FUNCTION_BLOCK basicFalhaFeedback (* Basic Function Block Type *)
  (* Standard: 61499-2 *)
  (* Version 0.0, 14/01/2026, Schneider Electric, Template *)
  PACKAGE Hidryco.HidrycoLib;
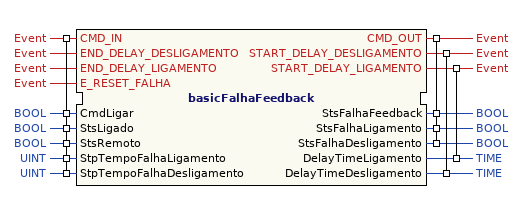
  EVENT_INPUT
    CMD_IN WITH StpTempoFalhaLigamento, StpTempoFalhaDesligamento, StsRemoto, CmdLigar, StsLigado;
    END_DELAY_DESLIGAMENTO; (* Normal Execution Request *)
    END_DELAY_LIGAMENTO;
    E_RESET_FALHA;
  END_EVENT
  EVENT_OUTPUT
    CMD_OUT WITH StsFalhaFeedback, StsFalhaLigamento, StsFalhaDesligamento;
    START_DELAY_DESLIGAMENTO WITH DelayTimeDesligamento; (* Execution Confirmation *)
    START_DELAY_LIGAMENTO WITH DelayTimeLigamento;
  END_EVENT
  VAR_INPUT
    CmdLigar : BOOL;
    StsLigado : BOOL;
    StsRemoto : BOOL;
    StpTempoFalhaLigamento : UINT;
    StpTempoFalhaDesligamento : UINT;
  END_VAR
  VAR_OUTPUT
    StsFalhaFeedback : BOOL;
    StsFalhaLigamento : BOOL;
    StsFalhaDesligamento : BOOL;
    DelayTimeLigamento : TIME;
    DelayTimeDesligamento : TIME;
  END_VAR
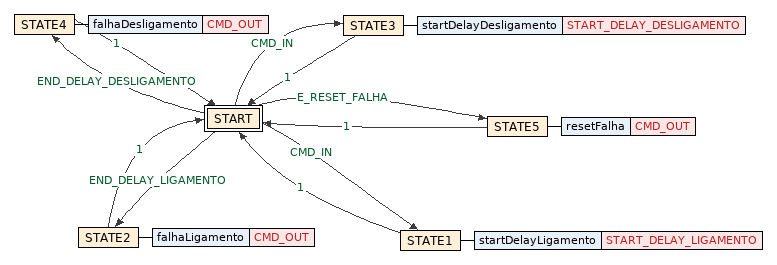
  EC_STATES
    START; (* Initial State *)
    STATE1 : startDelayLigamento -> START_DELAY_LIGAMENTO;
    STATE2 : falhaLigamento -> CMD_OUT;
    STATE3 : startDelayDesligamento -> START_DELAY_DESLIGAMENTO;
    STATE4 : falhaDesligamento -> CMD_OUT;
    STATE5 : resetFalha -> CMD_OUT;
  END_STATES
  EC_TRANSITIONS
    START TO STATE1 := CMD_IN;
    STATE1 TO START := 1;
    START TO STATE2 := END_DELAY_LIGAMENTO;
    STATE2 TO START := 1;
    START TO STATE3 := CMD_IN;
    STATE3 TO START := 1;
    START TO STATE4 := END_DELAY_DESLIGAMENTO;
    STATE4 TO START := 1;
    START TO STATE5 := E_RESET_FALHA;
    STATE5 TO START := 1;
  END_TRANSITIONS
  ALGORITHM falhaLigamento IN ST:
StsFalhaLigamento := 1;
StsFalhaFeedback := 1;
;
  END_ALGORITHM
  ALGORITHM falhaDesligamento IN ST:
StsFalhaDesligamento := 1;
StsFalhaFeedback := 1;
;
  END_ALGORITHM
  ALGORITHM resetFalha IN ST:
StsFalhaLigamento := 0;
StsFalhaDesligamento := 0;
StsFalhaFeedback := 0;
;
  END_ALGORITHM
  ALGORITHM startDelayLigamento IN ST:
IF (StsRemoto AND (NOT E_RESET_FALHA) AND CmdLigar AND (NOT StsLigado)) THEN
	DelayTimeLigamento := DINT_TO_TIME(UINT_TO_DINT(StpTempoFalhaLigamento) * 1000);
END_IF;
;
  END_ALGORITHM
  ALGORITHM startDelayDesligamento IN ST:
IF StsRemoto AND (NOT E_RESET_FALHA) AND (NOT CmdLigar) AND StsLigado THEN
	DelayTimeDesligamento := DINT_TO_TIME(UINT_TO_DINT(StpTempoFalhaDesligamento) * 1000);
END_IF;
;
  END_ALGORITHM
END_FUNCTION_BLOCK
